FUNCTION_BLOCK INTERNAL FB_AlarmManager_Tests EXTENDS FB_TestSuite
VAR_INPUT
END_VAR
VAR_OUTPUT
END_VAR
VAR;
	_alarmManager	: FB_AlarmManager(TRUE, 0);
	_alarmsArray	: ARRAY[0..100] OF ST_AlarmInfo;
	n				: T_ArrayIndexer;
END_VAR

_alarmManager(refAlarms := _alarmsArray);

Test00_RegisterAlarms();
Test01_ActivateNewAlarm_ExpectUnacknowledgedActiveAlarm();
Test02_AcknowledgeActiveAlarm_ExpectActiveAcknowledged();
Test03_ActivateExistingAlarm_ExpectSameActiveAlarmCount();
Test04_DeactivateAlarm_ExpectNotActiveAcknowledged();
Test05_AcknowlidgeInactiveAlarm_ExpectAcknowledgedNotActive();
Test06_DisableManager_ExpectNoActiveAlarms();
Test07_AcknowledgeAllAlarms_ExpectActiveAlarmsUnchanged();
Test08_ActivateByName();
Test09_DeactivateByName();
Test10_AcknowledgeByName();
Test11_GetAlarmByName();
Test12_GetAlarmById();
Test13_ActivateById();
Test14_DeactivateById();
Test15_AcknowledgeById();
Test16_TimeInfos();

METHOD Test00_RegisterAlarms
VAR_INPUT
END_VAR

VAR
	addAlarmIndex	: T_ArrayIndexer;
END_VAR
TcUnit.TEST('Test00_RegisterAlarms');
_alarmManager.Actions().Acknowledge();
AssertEquals_UDINT(
	Actual := _alarmManager.MaximumAlarmsCount,
	Expected := 101,
	Message := 'Total number of allowed alarms to be registered is incorrect.');

FOR addAlarmIndex := 1 TO 100 BY 1 DO
	AssertTrue(
		Condition := _alarmManager.RegisterAlarm(
			Id := addAlarmIndex,
			Message := CONCAT('Alarm message', TO_STRING(addAlarmIndex)),
			Name := CONCAT('Alarm name', TO_STRING(addAlarmIndex))),
		Message := 'Registering alarm failed.');
		
	AssertEquals_UDINT(
		Actual := _alarmManager.RegisteredAlarmsCount,
		Expected := DINT_TO_UDINT(addAlarmIndex),
		Message := 'Registered alarm count is incorrect.');
		
	AssertTrue(
		Condition := _alarmManager.GetAlarmById(nID := addAlarmIndex).IsAcknowledged,
		Message := 'Newly registered alarm should be acknowledged by default, when created.');
END_FOR


AssertFalse(
	Condition := _alarmManager.RegisterAlarm(
		Id := 22,
		Message := CONCAT('Alarm message', TO_STRING(addAlarmIndex - 1)),
		Name := CONCAT('Alarm name', TO_STRING(addAlarmIndex - 1))),
	Message := 'Registering an alarm with an existing id should not be possible.');

AssertTrue(
	Condition := _alarmManager.RegisterAlarm(
		Id := addAlarmIndex + 1,
		Message := CONCAT('Alarm message', TO_STRING(addAlarmIndex)),
		Name := CONCAT('Alarm name', TO_STRING(addAlarmIndex))),
	Message := 'Registering alarm failed.');
AssertEquals_UDINT(
	Actual := _alarmManager.RegisteredAlarmsCount,
	Expected := DINT_TO_UDINT(addAlarmIndex),
	Message := 'Registered alarm count is incorrect.');

AssertFalse(
	Condition := _alarmManager.RegisterAlarm(
		Id := 333,
		Message := CONCAT('Alarm message', TO_STRING(addAlarmIndex)),
		Name := CONCAT('Alarm name', TO_STRING(addAlarmIndex))),
	Message := 'Registering an alarm when the entire buffer has been filled should not be possible.');
	
TcUnit.TEST_FINISHED();
END_METHOD

METHOD Test01_ActivateNewAlarm_ExpectUnacknowledgedActiveAlarm
VAR_INPUT
END_VAR

VAR
	currentAlarm	: ST_AlarmInfo;
END_VAR
TcUnit.TEST('Test01_ActivateNewAlarm_ExpectUnacknowledgedActiveAlarm');

_alarmManager.RaiseAlarmById(10);
currentAlarm := _alarmManager.GetAlarmById(10);

AssertEquals_BOOL(
	Actual := currentAlarm.IsActive,
	Expected := TRUE,
	Message := 'Alarm activation failed.');
	
AssertEquals_BOOL(
	Actual := currentAlarm.IsAcknowledged,
	Expected := FALSE,
	Message := 'Newly activated alarm should not be acknowledged.');	

	
AssertEquals_UINT(
	Actual := _alarmManager.ActiveAlarmsCount,
	Expected := 1,
	Message := 'Active alarm count is incorrect.');

AssertEquals_UINT(
	Actual := _alarmManager.UnacknowledgedAlarmsCount,
	Expected := 1,
	Message := 'Unacknowledged alarm count is incorrect.');
	
TcUnit.TEST_FINISHED();
END_METHOD

METHOD Test02_AcknowledgeActiveAlarm_ExpectActiveAcknowledged
VAR_INPUT
END_VAR
TcUnit.TEST('Test02_AcknowledgeActiveAlarm_ExpectActiveAcknowledged');

_alarmManager.AcknowledgeAlarmById(10);

AssertEquals_BOOL(
	Actual := _alarmManager.GetAlarmById(10).IsActive,
	Expected := TRUE,
	Message := 'Alarm activation failed.');
	
AssertEquals_BOOL(
	Actual := _alarmManager.GetAlarmById(10).IsAcknowledged,
	Expected := TRUE,
	Message := 'Acknowlidging active alarm failed.');	

TcUnit.TEST_FINISHED();
END_METHOD

METHOD Test03_ActivateExistingAlarm_ExpectSameActiveAlarmCount
VAR_INPUT
END_VAR
TcUnit.TEST('Test03_ActivateExistingAlarm_ExpectSameActiveAlarmCount');

_alarmManager.RaiseAlarmById(10);
_alarmManager();

AssertEquals_BOOL(
	Actual := _alarmManager.GetAlarmById(10).IsActive,
	Expected := TRUE,
	Message := 'Alarm activation failed.');
	
AssertEquals_BOOL(
	Actual := _alarmManager.GetAlarmById(10).IsAcknowledged,
	Expected := TRUE,
	Message := 'Already acknowledged alarm should not be acknowledged when activating the alarm while it is already active.');	

	
AssertEquals_UINT(
	Actual := _alarmManager.ActiveAlarmsCount,
	Expected := 1,
	Message := 'Active alarm count is incorrect.');

AssertEquals_UINT(
	Actual := _alarmManager.UnacknowledgedAlarmsCount,
	Expected := 0,
	Message := 'Activating acknowledged and already active alarm should not cause the alarm to be unacknowledged..');
	
TcUnit.TEST_FINISHED();
END_METHOD

METHOD Test04_DeactivateAlarm_ExpectNotActiveAcknowledged
VAR_INPUT
END_VAR
TcUnit.TEST('Test04_DeactivateAlarm_ExpectNotActiveAcknowledged');

_alarmManager.DeactivateAlarmById(10);
_alarmManager();

AssertFalse(
	Condition := _alarmManager.GetAlarmById(10).IsActive,
	Message := 'Alarm deactivation failed.');
	
AssertTrue(
	Condition := _alarmManager.GetAlarmById(10).IsAcknowledged,
	Message := 'Alarm deactivation should not acknowledge the alarm.');	
	
AssertEquals_UINT(
	Actual := _alarmManager.ActiveAlarmsCount,
	Expected := 0,
	Message := 'Active alarm count is incorrect.');

AssertEquals_UINT(
	Actual := _alarmManager.UnacknowledgedAlarmsCount,
	Expected := 0,
	Message := 'Unacknowledged alarm count is incorrect.');
	
TcUnit.TEST_FINISHED();
END_METHOD

METHOD Test05_AcknowlidgeInactiveAlarm_ExpectAcknowledgedNotActive
VAR_INPUT
END_VAR
TcUnit.TEST('Test05_AcknowlidgeInactiveAlarm_ExpectAcknowledgedNotActive');

_alarmManager.AcknowledgeAlarmById(10);
_alarmManager();

AssertEquals_BOOL(
	Actual := _alarmManager.GetAlarmById(10).IsActive,
	Expected := FALSE,
	Message := 'Alarm deactivation failed.');
	
AssertEquals_BOOL(
	Actual := _alarmManager.GetAlarmById(10).IsAcknowledged,
	Expected := TRUE,
	Message := 'Acknowlidging alarm failed.');	

	
AssertEquals_UINT(
	Actual := _alarmManager.ActiveAlarmsCount,
	Expected := 0,
	Message := 'Active alarm count is incorrect.');

AssertEquals_UINT(
	Actual := _alarmManager.UnacknowledgedAlarmsCount,
	Expected := 0,
	Message := 'Unacknowledged alarm count is incorrect.');
	
TcUnit.TEST_FINISHED();
END_METHOD

METHOD Test06_DisableManager_ExpectNoActiveAlarms
VAR_INPUT
END_VAR
VAR
	n	: T_ArrayIndexer;
END_VAR
TcUnit.TEST('Test06_DisableManager_ExpectNoActiveAlarms');

FOR n := 1 TO 40 BY 1 DO
	_alarmManager.RaiseAlarmById(n);
END_FOR

AssertEquals_UINT(
	Expected := 40,
	Actual := _alarmManager.ActiveAlarmsCount,
	Message := 'There should only be 40 active alarms at this point.');
		
_alarmManager.Enable := FALSE;

AssertEquals_UINT(
	Expected := 0,
	Actual := _alarmManager.ActiveAlarmsCount,
	Message := 'Disabling the manager should result in all of the alarms being inactive.');

_alarmManager.Enable := TRUE;

TcUnit.TEST_FINISHED();
END_METHOD

METHOD Test07_AcknowledgeAllAlarms_ExpectActiveAlarmsUnchanged
VAR_INPUT
END_VAR

VAR
	n				: T_ArrayIndexer;
	fbAlarmManager	: FB_AlarmManager(TRUE, 0);
	arrAlarms		: ARRAY[0..60] OF ST_AlarmInfo;
END_VAR
TcUnit.TEST('Test07_AcknowledgeAllAlarms_ExpectActiveAlarmsUnchanged');

fbAlarmManager(refAlarms := arrAlarms);
FOR n := 1 TO 40 BY 1 DO
	fbAlarmManager.RegisterAlarm(n, TO_STRING(n), '');
	fbAlarmManager.RaiseAlarmById(n);
END_FOR

AssertEquals_UINT(
	Expected := 40,
	Actual := fbAlarmManager.ActiveAlarmsCount,
	Message := 'There should only be 40 active alarms at this point.');
		
fbAlarmManager.AcknowledgeAllAlarms();

AssertEquals_UINT(
	Expected := 0,
	Actual := fbAlarmManager.UnacknowledgedAlarmsCount,
	Message := 'Acknowlidging all alarms should result in no unacknowledged alarms.');

AssertEquals_UINT(
	Expected := 40,
	Actual := fbAlarmManager.ActiveAlarmsCount,
	Message := 'There should still be 40 active alarms, acknowlidning alarms should not affect alarm state.');


TcUnit.TEST_FINISHED();
END_METHOD

METHOD Test08_ActivateByName
VAR_INPUT
END_VAR
TcUnit.TEST('Test08_ActivateByName');

// Reset all alarms this way
_alarmManager.Enable := FALSE;
_alarmManager.Enable := TRUE;

_alarmManager.RaiseAlarmByName('Alarm name10');

AssertTrue(
	Condition := _alarmManager.GetAlarmByName('Alarm name10').IsActive,
	Message := 'Activating alarm by name failed.');

AssertFalse(
	Condition := _alarmManager.GetAlarmByName('Alarm name10').IsAcknowledged,
	Message := 'Alarm shold be unacknowledged.');
	
_alarmManager.DeactivateAlarmByName('Alarm name10');
_alarmManager.AcknowledgeAlarmByName('Alarm name10');

_alarmManager.Actions()
	.Raise()
	.ByName('Alarm name10');

AssertTrue(
	Condition := _alarmManager.GetAlarmByName('Alarm name10').IsActive,
	Message := 'Fluent - Activating alarm by name failed.');

AssertFalse(
	Condition := _alarmManager.GetAlarmByName('Alarm name10').IsAcknowledged,
	Message := 'Fluent - Alarm shold be unacknowledged.');
	
TcUnit.TEST_FINISHED();
END_METHOD

METHOD Test09_DeactivateByName
VAR_INPUT
END_VAR
TcUnit.TEST('Test09_DeactivateByName');

_alarmManager.DeactivateAlarmByName('Alarm name10');
AssertFalse(
	Condition := _alarmManager.GetAlarmByName('Alarm name10').IsActive,
	Message := 'Deactivate alarm by name failed.');

AssertFalse(
	Condition := _alarmManager.GetAlarmByName('Alarm name10').IsAcknowledged,
	Message := 'Alarm shold be unacknowledged.');
	
_alarmManager.RaiseAlarmByName('Alarm name10');
	
_alarmManager.Actions()
	.Deactivate()
	.ByName('Alarm name10');

AssertFalse(
	Condition := _alarmManager.GetAlarmByName('Alarm name10').IsActive,
	Message := 'Fluent - deactivating alarm by name failed.');

AssertFalse(
	Condition := _alarmManager.GetAlarmByName('Alarm name10').IsAcknowledged,
	Message := 'Fluent - Alarm shold be unacknowledged.');
	
TcUnit.TEST_FINISHED();
END_METHOD

METHOD Test10_AcknowledgeByName
VAR_INPUT
END_VAR
TcUnit.TEST('Test10_AcknowledgeByName');

_alarmManager.AcknowledgeAlarmByName('Alarm name10');

AssertTrue(
	Condition := _alarmManager.GetAlarmByName('Alarm name10').IsAcknowledged,
	Message := 'Alarm shold be acknowledged.');

	
_alarmManager.Actions().Raise().ByName('Alarm name10');
_alarmManager.Actions().Deactivate().ByName('Alarm name10');
_alarmManager.Actions().Acknowledge().ByName('Alarm name10');
AssertTrue(
	Condition := _alarmManager.GetAlarmByName('Alarm name10').IsAcknowledged,
	Message := 'Fluent - Alarm shold be acknowledged.');
	
TcUnit.TEST_FINISHED();
END_METHOD

METHOD Test11_GetAlarmByName
VAR_INPUT
END_VAR

VAR_INST
	fbAlarmManager	: FB_AlarmManager(TRUE, 0);
	alarms			: ARRAY[0..10] OF ST_AlarmInfo;
	i				: T_ArrayIndexer;
END_VAR
TcUnit.TEST('Test11_GetAlarmByName');
fbAlarmManager(refAlarms := alarms);

FOR i := 1 TO 11 BY 1 DO
	fbAlarmManager.RegisterAlarm(i, TO_STRING(i), '');
	AssertEquals_STRING(
		Actual := fbAlarmManager.GetAlarmByName(sName := TO_STRING(i)).Name,
		Expected := TO_STRING(i),
		Message := CONCAT('Getting alarm by name failed for alarm', TO_STRING(i)));	
END_FOR

TcUnit.TEST_FINISHED();
END_METHOD

METHOD Test12_GetAlarmById
VAR_INPUT
END_VAR
VAR_INST
	fbAlarmManager	: FB_AlarmManager(TRUE, 0);
	alarms			: ARRAY[0..10] OF ST_AlarmInfo;
	i				: T_ArrayIndexer;
END_VAR
TcUnit.TEST('Test12_GetAlarmById');
fbAlarmManager(refAlarms := alarms);

FOR i := 1 TO 11 BY 1 DO
	fbAlarmManager.RegisterAlarm(i, TO_STRING(i), '');
	AssertEquals_DINT(
		Actual := fbAlarmManager.GetAlarmById(i).Id,
		Expected := i,
		Message := CONCAT('Getting alarm by id failed for alarm', TO_STRING(i)));	
END_FOR

TcUnit.TEST_FINISHED();
END_METHOD

METHOD Test13_ActivateById
VAR_INPUT
END_VAR
TcUnit.TEST('Test13_ActivateById');

// Reset all alarms this way
_alarmManager.Enable := FALSE;
_alarmManager.Enable := TRUE;

_alarmManager.RaiseAlarmById(10);

AssertTrue(
	Condition := _alarmManager.GetAlarmById(10).IsActive,
	Message := 'Activating alarm by id failed.');

AssertFalse(
	Condition := _alarmManager.GetAlarmById(10).IsAcknowledged,
	Message := 'Alarm shold be unacknowledged.');
	
_alarmManager.DeactivateAlarmById(10);
_alarmManager.AcknowledgeAlarmById(10);

_alarmManager.Actions()
	.Raise()
	.ById(10);

AssertTrue(
	Condition := _alarmManager.GetAlarmById(10).IsActive,
	Message := 'Fluent - Activating alarm by name failed.');

AssertFalse(
	Condition := _alarmManager.GetAlarmById(10).IsAcknowledged,
	Message := 'Fluent - Alarm shold be unacknowledged.');
	
TcUnit.TEST_FINISHED();
END_METHOD

METHOD Test14_DeactivateById
VAR_INPUT
END_VAR
TcUnit.TEST('Test14_DeactivateById');

_alarmManager.DeactivateAlarmById(10);
AssertFalse(
	Condition := _alarmManager.GetAlarmById(10).IsActive,
	Message := 'Deactivate alarm by name failed.');

AssertFalse(
	Condition := _alarmManager.GetAlarmById(10).IsAcknowledged,
	Message := 'Alarm shold be unacknowledged.');
	
_alarmManager.RaiseAlarmById(13);
	
_alarmManager.Actions()
	.Deactivate()
	.ById(13);

AssertFalse(
	Condition := _alarmManager.GetAlarmById(10).IsActive,
	Message := 'Fluent - deactivating alarm by name failed.');

AssertFalse(
	Condition := _alarmManager.GetAlarmById(10).IsAcknowledged,
	Message := 'Fluent - Alarm shold be unacknowledged.');
	
TcUnit.TEST_FINISHED();
END_METHOD

METHOD Test15_AcknowledgeById
VAR_INPUT
END_VAR
TcUnit.TEST('Test15_AcknowledgeById');

_alarmManager.AcknowledgeAlarmById(10);

AssertTrue(
	Condition := _alarmManager.GetAlarmById(10).IsAcknowledged,
	Message := 'Alarm shold be acknowledged.');

	
_alarmManager.Actions().Raise().ById(10);
_alarmManager.Actions().Deactivate().ById(10);
_alarmManager.Actions().Acknowledge().ById(10);
AssertTrue(
	Condition := _alarmManager.GetAlarmById(10).IsAcknowledged,
	Message := 'Fluent - Alarm shold be acknowledged.');
	
TcUnit.TEST_FINISHED();
END_METHOD

METHOD Test16_TimeInfos
VAR_INPUT
END_VAR

VAR_INST
	fbAlarmManager			: FB_AlarmManager(TRUE, 0);
	alarms					: ARRAY[0..10] OF ST_AlarmInfo;
	i						: T_ArrayIndexer;
	stTimeStruct			: Tc2_Utilities.TIMESTRUCT;
	stTimeStructActivation	: Tc2_Utilities.TIMESTRUCT;	
	stTimeStructAcnowledge	: Tc2_Utilities.TIMESTRUCT;
	alarm			: ST_AlarmInfo;
END_VAR
TcUnit.TEST('Test16_TimeInfos');
fbAlarmManager(refAlarms := alarms);
IF fbAlarmManager._dateTime.CurrentTime.IsValid THEN
	FOR i := 0 TO 10 BY 1 DO
		fbAlarmManager.RegisterAlarm(i+1,'','');
		AssertEquals(
			Expected := stTimeStruct,
			Actual := fbAlarmManager.GetAlarmById(i).TimeInfos.Acknowledged,
			Message := 'Newly registered alarm should have empty time informations!');
		AssertEquals(
			Expected := stTimeStruct,
			Actual := fbAlarmManager.GetAlarmById(i).TimeInfos.Activated,
			Message := 'Newly registered alarm should have empty time informations!');
		AssertEquals(
			Expected := stTimeStruct,
			Actual := fbAlarmManager.GetAlarmById(i).TimeInfos.Deactivated,
			Message := 'Newly registered alarm should have empty time informations!');
	END_FOR
	
	// Raise alarm
	fbAlarmManager.Actions().Raise().ById(2);
	stTimeStruct := fbAlarmManager._dateTime.CurrentTime.Value;
	stTimeStructActivation := stTimeStruct;
	alarm := fbAlarmManager.GetAlarmById(2);
	AssertEquals_WORD(
		Expected := stTimeStruct.wMilliseconds,
		Actual := alarm.TimeInfos.Activated.wMilliseconds,
		Message := 'Activation time info after raising alarm (millisecond) is incorrect.');
	AssertEquals_WORD(
		Expected := stTimeStruct.wSecond,
		Actual := alarm.TimeInfos.Activated.wSecond,
		Message := 'Activation time info after raising alarm (second) is incorrect.');
	AssertEquals_WORD(
		Expected := stTimeStruct.wMinute,
		Actual := alarm.TimeInfos.Activated.wMinute,
		Message := 'Activation time info after raising alarm (minute) is incorrect.');
	AssertEquals_WORD(
		Expected := stTimeStruct.wHour,
		Actual := alarm.TimeInfos.Activated.wHour,
		Message := 'Activation time info after raising alarm (hour) is incorrect.');
	AssertEquals_WORD(
		Expected := stTimeStruct.wDay,
		Actual := alarm.TimeInfos.Activated.wDay,
		Message := 'Activation time info after raising alarm (day) is incorrect.');
	AssertEquals_WORD(
		Expected := stTimeStruct.wMonth,
		Actual := alarm.TimeInfos.Activated.wMonth,
		Message := 'Activation time info after raising alarm (month) is incorrect.');
	AssertEquals_WORD(
		Expected := stTimeStruct.wYear,
		Actual := alarm.TimeInfos.Activated.wYear,
		Message := 'Activation time info after raising alarm (year) is incorrect.');	
	AssertEquals_WORD(
		Expected := stTimeStruct.wDayOfWeek,
		Actual := alarm.TimeInfos.Activated.wDayOfWeek,
		Message := 'Activation time info after raising alarm (day of week) is incorrect.');
		
	MEMSET(ADR(stTimeStruct),0,SIZEOF(Tc2_Utilities.TIMESTRUCT));	
	AssertEquals(
		Expected := stTimeStruct,
		Actual := fbAlarmManager.GetAlarmById(2).TimeInfos.Acknowledged,
		Message := 'When alarm is raised, the acknowledged time information should be empty.');
	AssertEquals(
		Expected := stTimeStruct,
		Actual := fbAlarmManager.GetAlarmById(2).TimeInfos.Deactivated,
		Message := 'When alarm is raised, the deactivation time information should be empty.');
	
	// Acknowledge alarm
	fbAlarmManager.Actions().Acknowledge().ById(2);
	stTimeStruct := fbAlarmManager._dateTime.CurrentTime.Value;
	stTimeStructAcnowledge := stTimeStruct;
	alarm := fbAlarmManager.GetAlarmById(2);
	
	AssertEquals_WORD(
		Expected := stTimeStruct.wMilliseconds,
		Actual := alarm.TimeInfos.Acknowledged.wMilliseconds,
		Message := 'Acknowledged time info after acknowlidging alarm (millisecond) is incorrect.');
	AssertEquals_WORD(
		Expected := stTimeStruct.wSecond,
		Actual := alarm.TimeInfos.Acknowledged.wSecond,
		Message := 'Acknowledged time info after acknowlidging alarm (second) is incorrect.');
	AssertEquals_WORD(
		Expected := stTimeStruct.wMinute,
		Actual := alarm.TimeInfos.Acknowledged.wMinute,
		Message := 'Acknowledged time info after acknowlidging alarm (minute) is incorrect.');
	AssertEquals_WORD(
		Expected := stTimeStruct.wHour,
		Actual := alarm.TimeInfos.Acknowledged.wHour,
		Message := 'Acknowledged time info after acknowlidging alarm (hour) is incorrect.');
	AssertEquals_WORD(
		Expected := stTimeStruct.wDay,
		Actual := alarm.TimeInfos.Acknowledged.wDay,
		Message := 'Acknowledged time info after acknowlidging alarm (day) is incorrect.');
	AssertEquals_WORD(
		Expected := stTimeStruct.wMonth,
		Actual := alarm.TimeInfos.Acknowledged.wMonth,
		Message := 'Acknowledged time info after acknowlidging alarm (month) is incorrect.');
	AssertEquals_WORD(
		Expected := stTimeStruct.wYear,
		Actual := alarm.TimeInfos.Acknowledged.wYear,
		Message := 'Acknowledged time info after acknowlidging alarm (year) is incorrect.');	
	AssertEquals_WORD(
		Expected := stTimeStruct.wDayOfWeek,
		Actual := alarm.TimeInfos.Acknowledged.wDayOfWeek,
		Message := 'Acknowledged time info after acknowlidging alarm (day of week) is incorrect.');
	
	MEMSET(ADR(stTimeStruct),0,SIZEOF(Tc2_Utilities.TIMESTRUCT));	
	AssertEquals(
		Expected := stTimeStruct,
		Actual := fbAlarmManager.GetAlarmById(2).TimeInfos.Deactivated,
		Message := 'When alarm is acknowledged, the deactivation time information should not change.');
	AssertEquals(
		Actual := fbAlarmManager.GetAlarmById(2).TimeInfos.Activated,
		Expected := stTimeStructActivation,
		Message := 'If alarm is acknowledged, the acivation time info should not change.');
		
	// Deactivate alarm
	fbAlarmManager.Actions().Deactivate().ById(2);
	stTimeStruct := fbAlarmManager._dateTime.CurrentTime.Value;
	alarm := fbAlarmManager.GetAlarmById(2);
	
	AssertEquals_WORD(
		Expected := stTimeStruct.wMilliseconds,
		Actual := alarm.TimeInfos.Deactivated.wMilliseconds,
		Message := 'Deactivation time info after deactivating alarm (millisecond) is incorrect.');
	AssertEquals_WORD(
		Expected := stTimeStruct.wSecond,
		Actual := alarm.TimeInfos.Deactivated.wSecond,
		Message := 'Deactivation time info after deactivating alarm (second) is incorrect.');
	AssertEquals_WORD(
		Expected := stTimeStruct.wMinute,
		Actual := alarm.TimeInfos.Deactivated.wMinute,
		Message := 'Deactivation time info after deactivating alarm (minute) is incorrect.');
	AssertEquals_WORD(
		Expected := stTimeStruct.wHour,
		Actual := alarm.TimeInfos.Deactivated.wHour,
		Message := 'Deactivation time info after deactivating alarm (hour) is incorrect.');
	AssertEquals_WORD(
		Expected := stTimeStruct.wDay,
		Actual := alarm.TimeInfos.Deactivated.wDay,
		Message := 'Deactivation time info after deactivating alarm (day) is incorrect.');
	AssertEquals_WORD(
		Expected := stTimeStruct.wMonth,
		Actual := alarm.TimeInfos.Deactivated.wMonth,
		Message := 'Deactivation time info after deactivating alarm (month) is incorrect.');
	AssertEquals_WORD(
		Expected := stTimeStruct.wYear,
		Actual := alarm.TimeInfos.Deactivated.wYear,
		Message := 'Deactivation time info after deactivating alarm (year) is incorrect.');	
	AssertEquals_WORD(
		Expected := stTimeStruct.wDayOfWeek,
		Actual := alarm.TimeInfos.Deactivated.wDayOfWeek,
		Message := 'Deactivation time info after deactivating alarm (day of week) is incorrect.');
	
	// Check that previous entries did not change	
	AssertEquals(
		Expected := stTimeStructAcnowledge,
		Actual := fbAlarmManager.GetAlarmById(2).TimeInfos.Acknowledged,
		Message := 'When alarm is acknowledged, the deactivation time information should not change.');
	AssertEquals(
		Actual := fbAlarmManager.GetAlarmById(2).TimeInfos.Activated,
		Expected := stTimeStructActivation,
		Message := 'If alarm is acknowledged, the acivation time info should not change.');
	
		
	// Activate again and confirm that acknowledge and deactivation are reset
	// Raise alarm
	fbAlarmManager.Actions().Raise().ById(2);
	MEMSET(ADR(stTimeStruct),0,SIZEOF(Tc2_Utilities.TIMESTRUCT));
	AssertEquals(
		Actual := fbAlarmManager.GetAlarmById(2).TimeInfos.Deactivated,
		Expected := stTimeStruct,
		Message := 'When alarm is re-activated, previous time information for "deactivated" should be cleared.');
	AssertEquals(
		Actual := fbAlarmManager.GetAlarmById(2).TimeInfos.Acknowledged,
		Expected := stTimeStruct,
		Message := 'When alarm is re-activated, previous time information for "acknowledged" should be cleared.');
TcUnit.TEST_FINISHED();
END_IF
END_METHOD

END_FUNCTION_BLOCK

(* stored: Version 1.1.0.1, ProductVersion 3.1.4024.13
   POU FB_AlarmManager_Tests: Id {b130fb6f-8b4f-0495-3730-ec04c33d7bdb}, SpecialFunc None
   Method Test00_RegisterAlarms: Id {e3481e3b-1449-0574-29d8-60404d623878}
   Method Test01_ActivateNewAlarm_ExpectUnacknowledgedActiveAlarm: Id {9b1c592e-cc76-0bee-3ad8-28e7cb6b4bd3}
   Method Test02_AcknowledgeActiveAlarm_ExpectActiveAcknowledged: Id {7c9f10b9-d1cd-0984-3f11-39a43f41ca58}
   Method Test03_ActivateExistingAlarm_ExpectSameActiveAlarmCount: Id {10dfea8f-c6e2-0ed8-005c-f001e2b54921}
   Method Test04_DeactivateAlarm_ExpectNotActiveAcknowledged: Id {c90f406f-b4aa-00e6-3b58-9e9dd380a015}
   Method Test05_AcknowlidgeInactiveAlarm_ExpectAcknowledgedNotActive: Id {57171f97-e6ab-0277-376d-9e325dc8b13e}
   Method Test06_DisableManager_ExpectNoActiveAlarms: Id {61d52f1e-6c75-0a56-0857-ae9b851fb091}
   Method Test07_AcknowledgeAllAlarms_ExpectActiveAlarmsUnchanged: Id {b9eaba69-2f6e-05d7-364f-00d6655aa101}
   Method Test08_ActivateByName: Id {6570a093-9568-07a3-22a8-55d06cc88f21}
   Method Test09_DeactivateByName: Id {2a91d4bb-980f-0ce8-3024-53eef98592a9}
   Method Test10_AcknowledgeByName: Id {458fbcda-a528-09fc-3681-887d5d5998c3}
   Method Test11_GetAlarmByName: Id {96f09601-4dae-0dc0-2b2f-a3cb43f168d9}
   Method Test12_GetAlarmById: Id {cb3671fe-21bd-0cef-2a9f-51bdf7ac7e68}
   Method Test13_ActivateById: Id {22a01bfc-9e00-0fdb-0eb8-4a94e22c27b2}
   Method Test14_DeactivateById: Id {488d434c-be9c-0d2d-1a32-d0b1abb3bbf1}
   Method Test15_AcknowledgeById: Id {818eebe6-f990-0feb-303b-b323cafbcad0}
   Method Test16_TimeInfos: Id {7119724e-946e-01a5-10d2-4f0eba1adb0b} *)
